Staubli VAL3: start.pgx

program start()
  local num l_nError
  local num l_nKey
  local string l_sCaption
begin
  cls()
  userPage()
  // Load the EntryBox library
  call create("EntryBox\EBDefinition","",0,l_nError)
  if l_nError!=0
    popUpMsg(sErrorMessage)
  endIf
  //
  call getCaption(l_sCaption)
  // Set the default value of the boolean Textbox to TRUE
  call setFieldValue("Boolean :",pw:sTRUE,l_nError)
  if l_nError!=0
    popUpMsg(sErrorMessage)
  endIf
  // Display the EntryBox with a surrounding frame
  call display(1,1,true)
  // Manage the EntryBox
  call handle(l_nKey)
  popUpMsg("You have pressed function Key number "+toString("",l_nKey))
  //
  cls()
end
